INTERFACE I_Cyl_AtWork

PROPERTY P_AtWork : BOOL
GET
END_GET
END_PROPERTY

END_INTERFACE

(* stored: Version 1.1.0.1, ProductVersion 3.1.4024.6
   Itf I_Cyl_AtWork: Id {0d14d68b-edf3-03b6-1e28-d226068ca19b}
   Property P_AtWork: Id {842b13b8-9154-010f-0489-8d41ad85324b}
   Get Get: Id {d4f128a5-aabd-05ba-039f-26088ff3acb5} *)
